(**
This function block abstracts the Beckhoff EtherCAT terminal EL1144
*)
FUNCTION_BLOCK EL1144 IMPLEMENTS I_terminal_execution
VAR_INPUT
END_VAR
VAR_OUTPUT
	DI_channel_1 		: I_HAL_DI :=_channel_1;
	DI_channel_2 		: I_HAL_DI :=_channel_2;
	DI_channel_3 		: I_HAL_DI :=_channel_3;
	DI_channel_4 		: I_HAL_DI :=_channel_4;
END_VAR
VAR
	WcState_WcState			AT%I*: BOOL;
	WcState_InputToggle		AT%I*: BOOL;
	InfoData_State			AT%I*: UINT;
	
	Channel_1_Input         AT%I*: BOOL;
	Channel_2_Input         AT%I*: BOOL;
	Channel_3_Input         AT%I*: BOOL;
	Channel_4_Input         AT%I*: BOOL;
	
	_channel_1 : HAL_DI_Channel(channel_number:=1);
	_channel_2 : HAL_DI_Channel(channel_number:=2);
	_channel_3 : HAL_DI_Channel(channel_number:=3);
	_channel_4 : HAL_DI_Channel(channel_number:=4);
END_VAR
VAR CONSTANT	
    HARDWARE_REVSION : UINT:=19;
END_VAR


_channel_1.wcState:= NOT  WcState_WcState;
_channel_2.wcState:= NOT  WcState_WcState;
_channel_3.wcState:= NOT  WcState_WcState;
_channel_4.wcState:= NOT  WcState_WcState;

_channel_1();
_channel_2();
_channel_3();
_channel_4();

_channel_1.terminal_value:=Channel_1_Input;
_channel_2.terminal_value:=Channel_2_Input;
_channel_3.terminal_value:=Channel_3_Input;
_channel_4.terminal_value:=Channel_4_Input;

METHOD FB_init : BOOL
VAR_INPUT
	bInitRetains : BOOL; // if TRUE, the retain variables are initialized (warm start / cold start)
	bInCopyCode : BOOL;  // if TRUE, the instance afterwards gets moved into the copy code (online change)
	CoE_communication_handler: I_CoE_communication_handler;
END_VAR
END_METHOD

METHOD run : BOOL
VAR_INPUT
END_VAR
THIS^();
END_METHOD

END_FUNCTION_BLOCK

(* stored: Version 1.1.0.1, ProductVersion 3.1.4024.6
   POU EL1144: Id {7ffe0544-4efa-062a-1de7-cd9ac004744c}, SpecialFunc None
   Method FB_init: Id {0514e9d3-a161-07b2-3d11-995cde65d771}
   Method run: Id {a0c8ae01-de41-05bc-25d7-d04e4927d63d} *)
